FUNCTION_BLOCK Stage18 (* Template for a Basic Function Block Type *)
  (* Standard: 61499-2 *)
  (* Version 1.0, 2021-06-20, HP *)
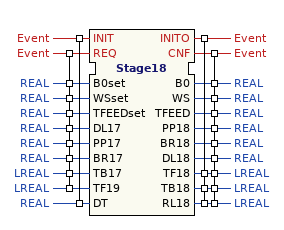
  EVENT_INPUT
    INIT WITH DT; (* Initialization Request *)
    REQ WITH B0set, WSset, TFEEDset, DL17, PP17, BR17, TB17, TF19; (* Normal Execution Request *)
  END_EVENT
  EVENT_OUTPUT
    INITO WITH TB18, RL18, TF18; (* Initialization Confirm *)
    CNF WITH TB18, DL18, TF18, BR18, PP18, B0, WS, TFEED, RL18; (* Execution Confirmation *)
  END_EVENT
  VAR_INPUT
    B0set : REAL;
    WSset : REAL;
    TFEEDset : REAL;
    DL17 : REAL;
    PP17 : REAL;
    BR17 : REAL;
    TB17 : LREAL;
    TF19 : LREAL;
    DT : REAL;
  END_VAR
  VAR_OUTPUT
    B0 : REAL;
    WS : REAL;
    TFEED : REAL;
    PP18 : REAL;
    BR18 : REAL;
    DL18 : REAL;
    TF18 : LREAL;
    TB18 : LREAL;
    RL18 : LREAL;
  END_VAR
  VAR
    AB : REAL; (* internal variabel *)
    UU : REAL;
    TREF : REAL;
    AD : REAL;
    AHC : REAL;
    AHR : REAL;
    AS : REAL;
    REC : REAL;
    WN : REAL;
    WN_1 : REAL;
    XKN : REAL;
    C1 : REAL;
    HS : REAL;
    G : REAL;
    W1 : REAL;
    TFREC : REAL;
    TS : REAL;
    DTS : REAL;
    TF18_last : REAL;
    RL18_last : REAL;
    TB18_last : REAL;
    USS : REAL;
    RHOB : REAL;
    CPB : REAL;
    CPF : REAL;
    FMW : REAL;
    HLV : REAL;
    HV : REAL;
    BPR : REAL;
    FMC : REAL;
    U : REAL;
    A : REAL;
    B : REAL;
    C : REAL;
    D1 : REAL;
    d : REAL;
    a : REAL;
    A1 : REAL;
    A2 : REAL;
    A3 : REAL;
    A4 : REAL;
    A5 : REAL;
    A6 : REAL;
    p : REAL;
    q : REAL;
    TC : REAL;
    PC : REAL;
    DTB18 : REAL;
    DEN18 : REAL;
    DH18 : REAL;
    DP18 : REAL;
    DPDH18 : REAL;
    DT18 : REAL;
    m : REAL;
    n : REAL;
    VR18 : REAL;
    DELTA18 : REAL;
    DELTA40 : REAL;
    DELTA62 : REAL;
    DELTA18_last : REAL;
    DELTA40_last : REAL;
    DELTA62_last : REAL;
  END_VAR
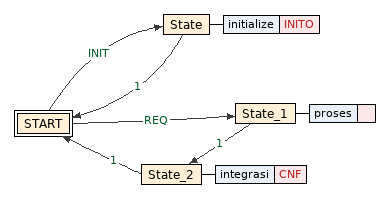
  EC_STATES
    START; (* Initial State *)
    State : initialize -> INITO;
    State_1 : proses;
    State_2 : integrasi -> CNF;
  END_STATES
  EC_TRANSITIONS
    START TO State := INIT;
    State TO START := 1;
    START TO State_1 := REQ;
    State_1 TO State_2 := 1;
    State_2 TO START := 1;
  END_TRANSITIONS
  ALGORITHM initialize IN ST: (* Initialization algorithm *)
TREF :=273.15;
AB :=57.2727;
AHC :=4069.2;
AHR :=2639.7;
AS :=3225.7;
REC :=0.0;
//TF2:=TF2;

//TFEED :=TFEED1+TREF;
 //TS:=TS1+TREF;
WN :=3.0;
XKN :=0.68;
HS:=0.11;
G :=9.81;
W1 :=0.50;

RL18 := 0.617636187854478;
TB18 := 321.44281037339;
TF18 := 318.266914942048;
TF19 := 316.357381861072;


RL18_last :=RL18;
TB18_last :=TB18;
TF18_last :=TF18;
  END_ALGORITHM
  ALGORITHM proses IN ST: (* kalkulasi *)
B0 :=B0set;
WS :=WSset;
TFEED:=TFEEDset;
UU := TFEEDset;
U :=UU;

USS :=49.767;
C1 :=0.625;
RHOB :=1032.4; //maassa jenis brine
CPB :=1.00; //heatcapacity Brine
CPF :=1.00; //heat capacity feed
FMW :=23654.0;
HLV :=563.7959;
HV :=625.1971;
BPR :=2.192;
FMC :=34736.09;
//U :=UU; //feed temp



///  Calculate the physical properties

//A :=3.2437814;
//B :=5.86826*0.001;
//C :=1.1702379*0.00000001;
//D1 :=2.1878462*0.001;
//TC :=647.27;
//PC :=218.167;


A1 :=3.2437814;
A2:=5.86826*0.001;
A3:=1.1702379*0.00000001;
A4 :=2.1878462*0.001;
A5 :=647.27;
A6 :=218.167;

DTB18 :=A5-TB18;
DEN18 :=(A1+A2*DTB18+A3*DTB18*DTB18*DTB18)/(1+A4*DTB18)*DTB18/TB18;
p:=DEN18;
q:=10.0;
PP18 :=A6/(EXPT(q, p));

// calculate the brine flow rates
DP18:=PP17-PP18;
DH18:=RL18-C1*HS;
DPDH18 :=DP18*101000+G*RHOB*DH18;
m:=DPDH18*RHOB;
n:=0.5;
BR18 :=WN*XKN*RL18*(EXPT(m, n));
BR18 :=BR18*60.0/1000.0;

// calculate the vapor flow rates

DT18 :=TB18-BPR/1.8-(TF19+TF18)*0.5;
VR18:=U*AHC*DT18/HLV/1000.0;
DL18 :=DL17+VR18;


//// state equation
DELTA18 :=(BR17-BR18-VR18)*1000.0/RHOB/AB;
DELTA40 :=((BR17*CPB*(TB17-TB18))-VR18*(HV-CPB*(TB18-TREF)))*1000.0/AB/RHOB/CPB/RL18;
DELTA62 :=(B0*CPF*(TF19-TF18)*1000+(U*AHC*DT18))/FMW/CPF;
  END_ALGORITHM
  ALGORITHM integrasi IN ST: (* new algorithm *)
B0 :=B0set;
WS :=WSset;
TFEED:=TFEEDset;
//integrasi
RL18 := (DELTA18 + DELTA18_last)*0.5*DT + RL18_last;
DELTA18_last :=DELTA18 ;
RL18_last :=RL18;

TB18:= (DELTA40 + DELTA40_last)*0.5*DT + TB18_last;
DELTA40_last :=DELTA40 ;
TB18_last:=TB18;

TF18 := (DELTA62 + DELTA62_last)*0.5*DT + TF18_last;
DELTA62_last :=DELTA62 ;
TF18_last :=TF18;
  END_ALGORITHM
END_FUNCTION_BLOCK
